# EPICS alarm handler configuration: mps_database/bare/alarms/areas/mpln_ltus_mp02.alhConfig
GROUP NULL MPLN:LTUS:MP02:1
$ALIAS MPS Link Node 204
$GUIDANCE
LTUH MPS
   Group Name: MPLN:LTUS:MP02:1
   Summary PV:  MPLN:LTUS:MP02:1:STATSUMY
$END
CHANNEL  MPLN:LTUS:MP02:1    MPLN:LTUS:MP02:1:MPS_EN_RBV		-----
CHANNEL  MPLN:LTUS:MP02:1    MPLN:LTUS:MP02:1:LC1_MODE_RBV		-----
